Fanuc KAREL source: ASIN.kl

PROGRAM T
%NOLOCKGROUP
VAR
 v0 : REAL
 res : REAL
BEGIN
 res = ASIN(v0)
END T
